TYPE ST_XPU_STRINGS :
STRUCT
  sXpuState       ,
  sXpuResult      ,
  sXpuCyclicCheck ,
  sXpuOpMode      ,
  sXpuMoverId_DetectionMode,
  sXpuMoverPosAssignement : STRING(30) := 'NULL';
END_STRUCT
END_TYPE

(* stored: Version 1.1.0.1, ProductVersion 3.1.4026.18
   DUT ST_XPU_STRINGS: Id {d072f511-f67c-4332-8a92-8b4239228af7} *)
